(* CODESYS project EZS1_Finished.project

Project tree, tasks and I/O mapping:
  Device : Berghof PPC V3 Control, Berghof Automation GmbH, version 3.12.3.0
    application Application
      libraries: Standard, * (System)
      task MainTask (cyclic, interval 4000 µs, priority 0) calls EtherCAT_Master.EtherCAT_Task [EtherCAT_Master.EtherCAT_Task], MAIN
      task EtherCAT_Task (cyclic, interval 4000 µs, priority 0) calls EtherCAT_Master.EtherCAT_Task [EtherCAT_Master.EtherCAT_Task]
      program MAIN [ST]
      program Simulation [ST]
      global variables Globale_Variablen
      visualisation DRUCKZYLINDER
      program Steuerung [FBD]
      program SSteuerungin [FBD]
      program SteuerungPOU [LD]
    EtherCAT_Master : EtherCAT Master, 3S - Smart Software Solutions GmbH, version 3.5.8.40
        settings: NetworkName = 'eth1'; NetworkName = "eth1"; SelectNetworkByName = True
      onboard_Buskoppler : onboard Buscoupler, Berghof Automation GmbH, version Revision=16#00000001
          settings: DC sync0 cycletime = 4000; DC sync1 cycletime = 4000
        E_I_O_DI16_DO16 : DI16/DO16 1ms 0.5A (204 800 100), Berghof Automation GmbH, version Revision=16#00000001
            settings: DC sync0 cycletime = 4000; DC sync1 cycletime = 4000
            unmapped channels: DigitalOutput0, DigitalOutput1, DigitalOutput2, DigitalOutput3, DigitalOutput4, DigitalOutput5, DigitalOutput6, DigitalOutput7, DigitalOutput8, DigitalOutput9, DigitalOutput10, DigitalOutput11, DigitalOutput12, DigitalOutput13, DigitalOutput14, DigitalOutput15, DigitalInput0, DigitalInput1, DigitalInput2, DigitalInput3, DigitalInput4, DigitalInput5, DigitalInput6, DigitalInput7, DigitalInput8, DigitalInput9, DigitalInput10, DigitalInput11, DigitalInput12, DigitalInput13, DigitalInput14, DigitalInput15
  text list GlobalTextList
*)

// Device/Application/Globale_Variablen
VAR_GLOBAL
	
	(* ------ Studenten-Variablen ------ *)
	(* --------------------------------- *)

	(* Ventile *) 
	V1 AT %QX0.0: BOOL;
	V2 AT %QX0.1: BOOL;
	V3 AT %QX0.2: BOOL;
	V4 AT %QX0.3: BOOL;
	
	(* Sensoren *)
	S1: BOOL;
	S2: BOOL;
 
	(* ------ Studenten-Variablen ENDE ------ *)
	(* -------------------------------------- *)
	
	S1_R AT %IX0.0: BOOL;
	S2_R AT %IX0.1: BOOL;

	
	(* Variablen zur Simulation *)
	(* ------------------------ *) 
	
	(* Reset & Co *) 
	RESET: BOOL := TRUE; 
	SIMULATION_ON: BOOL := TRUE;
	SIMULATION_OFF: BOOL := FALSE;
	
	(* Druck (konst.) *)
	Pinput: REAL;
	Poutside: REAL;
	
	(* DRUCK (var.) *)
	Pa: REAL;
	Pb: REAL;
	Pmanual: REAL := 0;
	
	(* Position des Zylinders *) 
	Xpos: REAL;
	MaxXpos: REAL;
	MinXpos: REAL;
	P2PosFaktor: REAL;
	
	(* Variablen fuer die Visualisierung *) 
	
	Draft: BOOL := FALSE;
	NotDraft: BOOL;
	
	Xpos4Vis: REAL := 0;
	V1_Vis: INT := 0;
	V2_Vis: INT := 0; 
	V3_Vis: INT := 0;
	V4_Vis: INT := 0;
	
	pull: BOOL := FALSE; 
	push: BOOL := FALSE; 

	STEUERUNG_ON: BOOL := FALSE;
END_VAR

// Device/Application/MAIN
PROGRAM MAIN
VAR
END_VAR

(* ------------------------------------- *)
(* --------- Studentenbereich ---------- *)

(* Aufgabe:
Erstellen Sie ein PRG 'Steuerung' dem Aufgabenblatt entsprechhend.
Benutzen Sie von den globalen Variablen NUR V1 - V4 und S1, S2.
Aktivieren Sie danach folgende Zeilen: 
*)

IF STEUERUNG_ON THEN
	SteuerungPOU();
END_IF; 

(* ------- ENDE Studentenbereich -------- *) 
(* -------------------------------------- *) 
(* Setze Durchzug *) 
(* -------------- *) 
IF ( (V1 AND V3) OR (V2 AND V4) )  THEN 
	Draft := TRUE; 
	NotDraft := FALSE; 
ELSE 
	Draft := FALSE; 
	NotDraft := TRUE; 
END_IF

(* Starte Simulation *) 
(* ----------------- *) 

IF SIMULATION_ON THEN 
	Simulation(); 
	SIMULATION_OFF := FALSE; 
	SIMULATION_ON := TRUE; 

ELSE 
	SIMULATION_OFF := TRUE; 
	SIMULATION_ON := FALSE; 
	
	S1 := S1_R;
	S2 := S2_R;
 
	IF ( S1 AND (NOT S2)) THEN
		Xpos := MaxXpos;
	ELSIF ((NOT S1) AND S2 ) THEN 
		Xpos := MinXpos;
	ELSE 
		Xpos := (MaxXpos-MinXpos)/2;
	END_IF
END_IF


(* Uebernehme die neue Position fuer die Visualisierung *)
(* ---------------------------------------------------- *) 
Xpos4Vis := -2.5*Xpos;

(* Aktualisiere die Visualisierung der Ventile *) 
(* ------------------------------------------- *)
IF V1 THEN V1_Vis := 40; ELSE V1_Vis := 0; END_IF;
IF V2 THEN V2_Vis := 40; ELSE V2_Vis := 0; END_IF; 
IF V3 THEN V3_Vis := 40; ELSE V3_Vis := 0; END_IF;
IF V4 THEN V4_Vis := 40; ELSE V4_Vis := 0; END_IF;

END_PROGRAM

// Device/Application/Steuerung
PROGRAM Steuerung
VAR
	Oben: BOOL;
	Oben_SR: SR;
END_VAR
VAR // added by the converter: edge detectors and wires of the graphical bodies
    _w1 : BOOL;
END_VAR

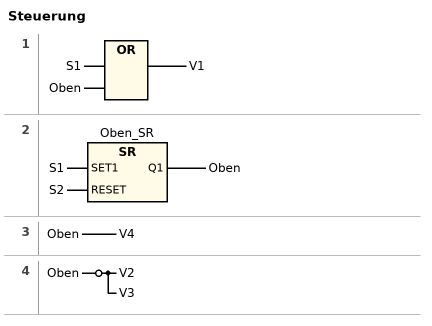
// NETWORK 1
V1 := S1 OR Oben;

// NETWORK 2
Oben_SR(SET1 := S1, RESET := S2); // SR
Oben := Oben_SR.Q1;

// NETWORK 3
V4 := Oben;

// NETWORK 4
_w1 := NOT Oben;
V2 := _w1;
V3 := _w1;

END_PROGRAM

// Device/Application/SteuerungPOU
PROGRAM SteuerungPOU
VAR
	schliessen: BOOL;
	TON_0: TON;
	RS_5: BOOL;
	S_5: BOOL;
	Entriegeltt: BOOL;
	open: BOOL;
	S1_in: BOOL;
	S2_in: BOOL;
	S1_out: INT;
	close: BOOL;
	unlock: BOOL;
	Cose_timer: TON;
	s5time: TIME:=T#5000MS;
	et: TIME;
	time_close: BOOL;
	block_timer: TON;
	blocked: BOOL;
	block: BOOL;
END_VAR

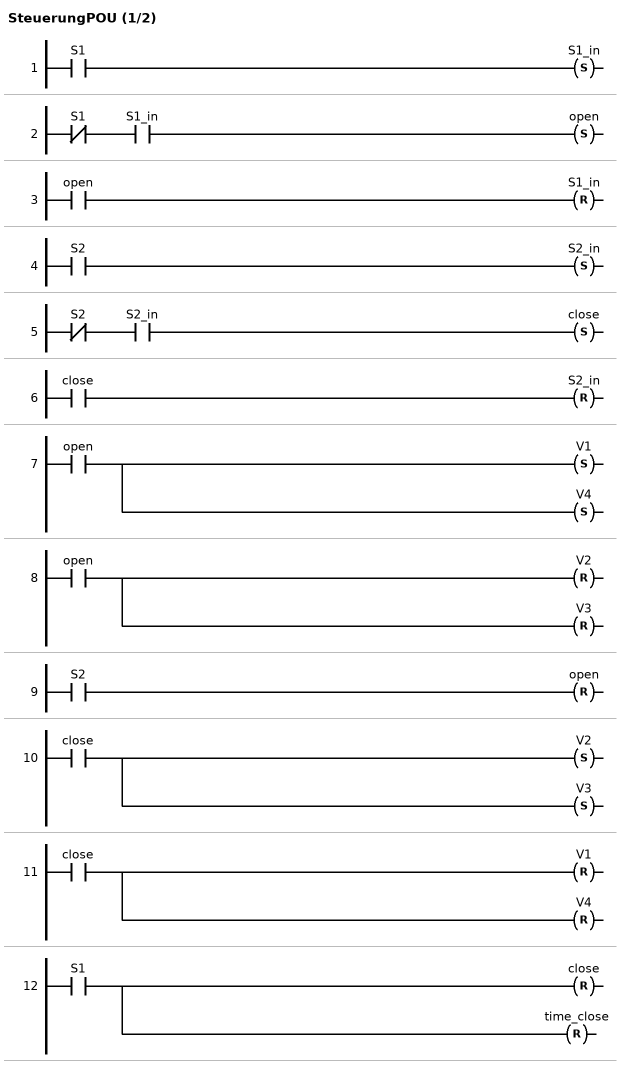
// NETWORK 1
S1_in S= S1;

// NETWORK 2
open S= NOT S1 AND S1_in;

// NETWORK 3
S1_in R= open;

// NETWORK 4
S2_in S= S2;

// NETWORK 5
close S= NOT S2 AND S2_in;

// NETWORK 6
S2_in R= close;

// NETWORK 7
V1 S= open;
V4 S= open;

// NETWORK 8
V2 R= open;
V3 R= open;

// NETWORK 9
open R= S2;

// NETWORK 10
V2 S= close;
V3 S= close;

// NETWORK 11
V1 R= close;
V4 R= close;

// NETWORK 12
close R= S1;
time_close R= S1;

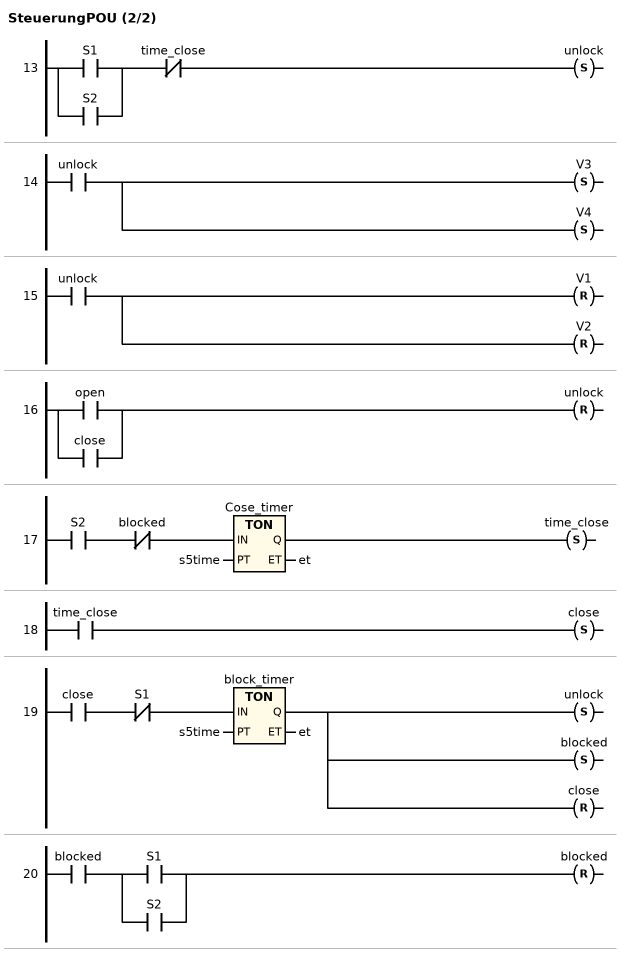
// NETWORK 13
unlock S= (S1 OR S2) AND NOT time_close;

// NETWORK 14
V3 S= unlock;
V4 S= unlock;

// NETWORK 15
V1 R= unlock;
V2 R= unlock;

// NETWORK 16
unlock R= open OR close;

// NETWORK 17
Cose_timer(IN := S2 AND NOT blocked, PT := s5time, ET => et); // TON
time_close S= Cose_timer.Q;

// NETWORK 18
close S= time_close;

// NETWORK 19
block_timer(IN := close AND NOT S1, PT := s5time, ET => et); // TON
unlock S= block_timer.Q;
blocked S= block_timer.Q;
close R= block_timer.Q;

// NETWORK 20
blocked R= blocked AND (S1 OR S2);

END_PROGRAM

// Device/Application/Simulation
PROGRAM Simulation
VAR
	DeltaXpos: REAL;
	NewXpos: REAL;
	RestVolumen: REAL := 1; 
END_VAR

(* INIT *) 
IF RESET THEN 
	(* Globale Konstanten festlegen*)
	Pinput := 2; 
	Poutside := 1; 
	P2PosFaktor := 2;  
	MaxXpos := 100; 
	MinXpos := 0; 
	
	(* Initialisiere den Druck, die Ventile und die Kolbenposition*)
	Pa := 1; 
	Pb := 1; 
	Pmanual := 0; 
	V1 := FALSE; 
	V2 := FALSE; 
	V3 := FALSE; 
	V4 := FALSE; 
	Xpos := 0; 
	
	RESET := FALSE;
 
ELSIF NotDraft THEN
	(* Aktualisiere manuellen Druck (ziehen oder druecken)*)
	IF (push AND (NOT pull)) THEN
		Pmanual := -1; 
	ELSIF ((NOT push) AND pull) THEN 
		Pmanual := 1; 
	ELSE 
		Pmanual := 0; 
	END_IF
	
	(* Bestimme die Verschiebung des Zylinders aus dem Druckunterschied *)
	DeltaXpos := (Pb - Pa+Pmanual)*P2PosFaktor;
	
	(* Bestimme die neue Position des Zylinders *)
	NewXpos := Xpos + DeltaXpos;
	IF ( NewXpos > MaxXpos ) THEN
		NewXPos := MaxXpos;
	ELSIF (NewXpos < MinXpos) THEN 
		NewXPos := MinXpos;  
	END_IF
	
	(* Aktualisiere den Druck P_alpha *) 
	IF ( V1 AND (NOT V3) ) THEN (* stabile Verbindung zur Druckluft => Druck entspricht P_input *) 
		IF NOT Draft THEN
			Pa := Pinput; 
		ELSE 
			Pa := Poutside; 
		END_IF
	ELSIF ( (NOT V1) AND V3) THEN (* stabile Verbindung nach draussen => Druck entspricht P_outside *) 
		Pa := Poutside; 
	ELSIF ( V1 AND V3 ) THEN (* Durchzug! Druckluft wird direkt nach draussen geleitet *) 
		Pa := Poutside; 
	ELSE (* Zylinderseite ist abgeschlossen => Druck wird an das Volumen angepasst *) 
		Pa := Pa * (MaxXpos - Xpos + RestVolumen) / (MaxXpos - NewXpos + RestVolumen); 
	END_IF
	
	(*Aktualisiere den Druck P_beta *) 
	IF ( V2 AND (NOT V4) ) THEN (* stabile Verbindung zur Druckluft => Druckluft entsprichht P_input *)
		IF NOT Draft THEN 
			Pb := Pinput;
		ELSE 
			Pb := Poutside; 
		END_IF
		
	ELSIF ( (NOT V2) AND V4 ) THEN (* stabile Verbindung nach draussen => Druck entspricht P_outside *) 
		Pb := Poutside; 
	ELSIF ( V2 AND V4) THEN (* Durchzug! Druckluft wird direkt nach draussen geleitet *) 
		Pb := Poutside; 
	ELSE (* Zylinderseite ist abgeschlossen => Druck  wird an das Volumen angepasst *)  
		Pb := Pb * (Xpos + Restvolumen) / (NewXpos + RestVolumen); 
	END_IF
	
	(* Uebernehme die neue Position *)
	Xpos := NewXpos; 
	
	(* Aktualisiere die Sensoren *)
	S1 := (Xpos >= MaxXpos-1);
	S2 := (Xpos <= MinXpos+1); 

END_IF

END_PROGRAM

// Device/Application/SSteuerungin
PROGRAM  SSteuerungin
VAR
	Unten: BOOL;
	Oben: BOOL;
	open: BOOL;
	close: BOOL;
	RS_0: RS;
	R_TRIG_0: R_TRIG;
	start_close: R_TRIG;
	end_close: F_TRIG;
	closing: R_TRIG;
	openall: F_TRIG;
	c: BOOL;
	start_open: R_TRIG;
	startclose: SR;
	startopen: SR;
	open_all: R_TRIG;
	SR_0: SR;
	RS_1: RS;
	RS_2: RS;
	RS_3: SR;
	RS_4: RS;
END_VAR

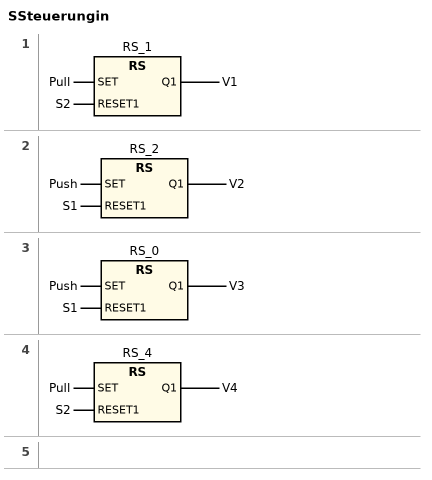
// NETWORK 1
RS_1(SET := Pull, RESET1 := S2); // RS
V1 := RS_1.Q1;

// NETWORK 2
RS_2(SET := Push, RESET1 := S1); // RS
V2 := RS_2.Q1;

// NETWORK 3
RS_0(SET := Push, RESET1 := S1); // RS
V3 := RS_0.Q1;

// NETWORK 4
RS_4(SET := Pull, RESET1 := S2); // RS
V4 := RS_4.Q1;

// NETWORK 5

END_PROGRAM

// Device/Application/DRUCKZYLINDER
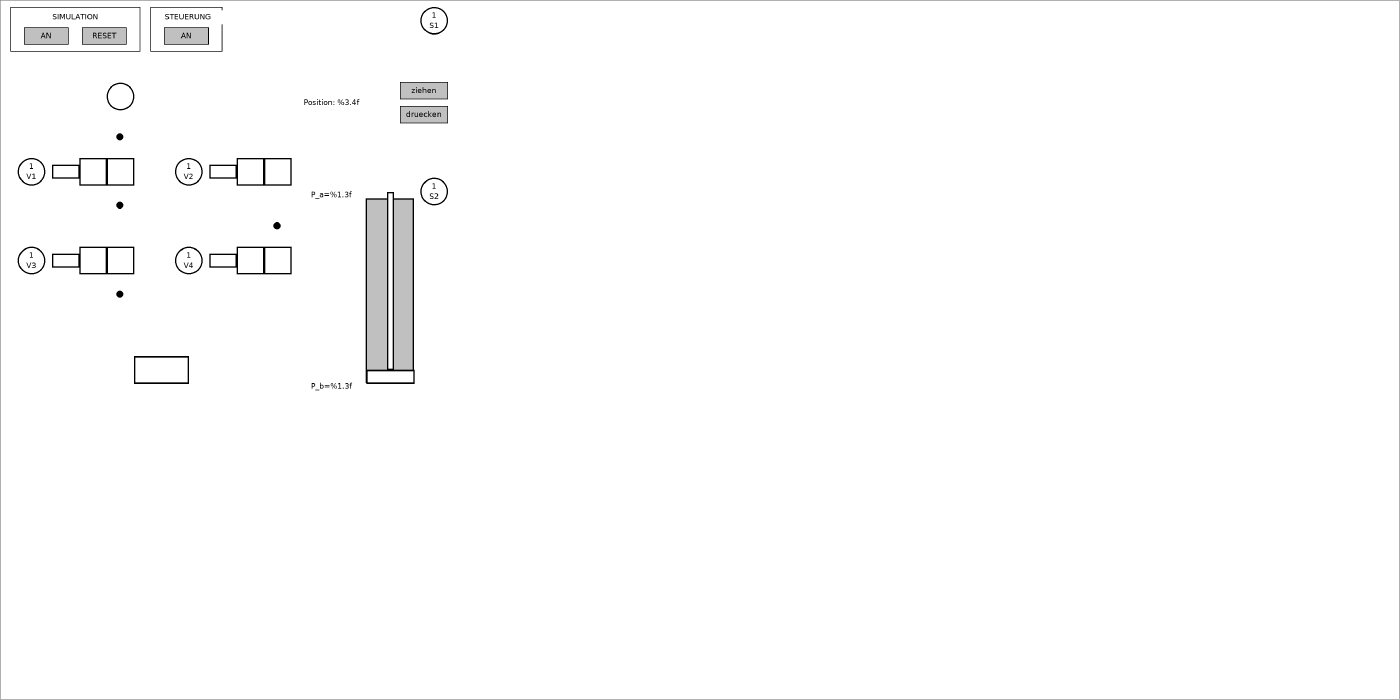
VISUALIZATION DRUCKZYLINDER  // 2048x1024
    Rectangle (220,10 105x65)
    Rectangle (15,10 190x65)
    Rectangle (60,15 100x20), "SIMULATION"
    Rectangle (535,290 70x270)
    Ellipse (615,10 40x40), colour toggle: Globale_Variablen.S1
    Ellipse (615,260 40x40), colour toggle: Globale_Variablen.S2
    Rectangle (440,275 90x20), "P_a=%1.3f", text variable: Globale_Variablen.Pa, invisible if: Globale_Variablen.SIMULATION_OFF
    Rectangle (440,555 90x20), "P_b=%1.3f", text variable: Globale_Variablen.Pb, invisible if: Globale_Variablen.SIMULATION_OFF
    Rectangle (425,140 120x20), "Position: %3.4f", text variable: Globale_Variablen.Xpos, invisible if: Globale_Variablen.SIMULATION_OFF
    RoundedRectangle (120,40 65x25), "RESET", colour toggle: Globale_Variablen.RESET
        toggle Globale_Variablen.RESET
    Group (536,281 68x278)
        p2738717112: Globale_Variablen.Xpos4Vis
        Rectangle (30,0 10x260)
        Rectangle (0,260 70x20)
    Polygon (535,310)
    Polygon (535,560)
    Polygon (535,310)
    Rectangle (615,30 40x15), "S1"
    Rectangle (615,15 40x15), "1"
    Rectangle (615,280 40x15), "S2"
    Rectangle (615,265 40x15), "1"
    Polyline (655,280)
    Polyline (655,30)
    Polyline (175,230)
    Group (131,121 63x38)
        Rectangle (0,15 30x10)
        Polyline (30,15)
        Polyline (30,25)
        Ellipse (25,0 40x40)
        Polygon (45,40)
    Group (26,231 118x38), input disabled if: Globale_Variablen.SIMULATION_OFF
        toggle Globale_Variablen.V1
        Polyline (120,20)
        Ellipse (0,0 40x40), colour toggle: Globale_Variablen.V1
            toggle Globale_Variablen.V1
        Rectangle (0,5 40x15), "1"
        Polyline (60,20)
        Rectangle (0,20 40x15), "V1"
    Group (76,231 118x38)
        p3560616238: Globale_Variablen.V1_Vis
        Rectangle (0,10 40x20)
        Rectangle (40,0 40x40)
        Rectangle (80,0 40x40)
        Polyline (100,10)
        Polyline (100,40)
        Polyline (105,10)
        Polyline (105,30)
        Polyline (60,40)
        Polygon (55,25)
        Polygon (15,30)
    Group (26,361 118x38), input disabled if: Globale_Variablen.SIMULATION_OFF
        toggle Globale_Variablen.V3
        Polyline (120,20)
        Ellipse (0,0 40x40), colour toggle: Globale_Variablen.V3
            toggle Globale_Variablen.V3
        Rectangle (0,5 40x15), "1"
        Polyline (60,20)
        Rectangle (0,20 40x15), "V3"
    Group (256,361 118x38), input disabled if: Globale_Variablen.SIMULATION_OFF
        toggle Globale_Variablen.V4
        Polyline (120,20)
        Ellipse (0,0 40x40), colour toggle: Globale_Variablen.V4
            toggle Globale_Variablen.V4
        Rectangle (0,5 40x15), "1"
        Polyline (60,20)
        Rectangle (0,20 40x15), "V4"
    Group (256,231 118x38), input disabled if: Globale_Variablen.SIMULATION_OFF
        toggle Globale_Variablen.V2
        Polyline (120,20)
        Ellipse (0,0 40x40), colour toggle: Globale_Variablen.V2
            toggle Globale_Variablen.V2
        Rectangle (0,5 40x15), "1"
        Polyline (60,20)
        Rectangle (0,20 40x15), "V2"
    Group (76,361 118x38)
        p3560616238: Globale_Variablen.V3_Vis
        Rectangle (0,10 40x20)
        Rectangle (40,0 40x40)
        Rectangle (80,0 40x40)
        Polyline (100,10)
        Polyline (100,40)
        Polyline (105,10)
        Polyline (105,30)
        Polyline (60,40)
        Polygon (55,25)
        Polygon (15,30)
    Group (306,231 118x38)
        p3560616238: Globale_Variablen.V2_Vis
        Rectangle (0,10 40x20)
        Rectangle (40,0 40x40)
        Rectangle (80,0 40x40)
        Polyline (100,10)
        Polyline (100,40)
        Polyline (105,10)
        Polyline (105,30)
        Polyline (60,40)
        Polygon (55,25)
        Polygon (15,30)
    Polyline (175,360)
    Polyline (405,360)
    Polyline (405,230)
    Polyline (535,300)
    Ellipse (170,195 10x10)
    Polyline (405,430)
    Polyline (485,330)
    Ellipse (170,295 10x10)
    Polyline (405,200)
    Ellipse (400,325 10x10)
    Polyline (485,550)
    Polyline (535,550)
    Ellipse (170,425 10x10)
    Polyline (405,430)
    Polyline (175,540)
    Group (196,521 93x38)
        Rectangle (0,0 80x40), colour toggle: Globale_Variablen.Draft
        Polygon (80,30)
        Polyline (20,0)
        Polyline (40,10)
        Polyline (60,0)
    Group (276,456 73x73), invisible if: Globale_Variablen.NotDraft
        Ellipse (20,15 30x30)
        Ellipse (35,25 30x30)
        Ellipse (5,10 30x30)
        Ellipse (25,0 30x30)
        Ellipse (45,10 30x30)
        Polygon (0,75)
    Polyline (195,540)
    Group (306,361 118x38)
        p3560616238: Globale_Variablen.V4_Vis
        Rectangle (0,10 40x20)
        Rectangle (40,0 40x40)
        Rectangle (80,0 40x40)
        Polyline (100,10)
        Polyline (100,40)
        Polyline (105,10)
        Polyline (105,30)
        Polyline (60,40)
        Polygon (55,25)
        Polygon (15,30)
    RoundedRectangle (585,120 70x25), "ziehen", colour toggle: Globale_Variablen.pull, invisible if: Globale_Variablen.SIMULATION_OFF, input disabled if: Globale_Variablen.SIMULATION_OFF
        tap Globale_Variablen.pull
    RoundedRectangle (585,155 70x25), "druecken", colour toggle: Globale_Variablen.push, invisible if: Globale_Variablen.SIMULATION_OFF, input disabled if: Globale_Variablen.SIMULATION_OFF
        tap Globale_Variablen.push
    RoundedRectangle (35,40 65x25), "AN", colour toggle: Globale_Variablen.SIMULATION_ON
        toggle Globale_Variablen.SIMULATION_ON
    RoundedRectangle (240,40 65x25), "AN", colour toggle: Globale_Variablen.STEUERUNG_ON
        toggle Globale_Variablen.STEUERUNG_ON
    Rectangle (225,15 100x20), "STEUERUNG"
END_VISUALIZATION
